// TIA Portal project "SimpleProject" (V17)

(* hardware
DEVICE "PLC_1"  S7-1200 Station
   slot 0: "Rack_0"  S7-1200 Rack  Rack  V1.0
   slot 1: "PLC_1"  CPU 1214C AC/DC/Rly  6ES7 214-1BG40-0XB0  V4.5
*)

// ===== PLC "PLC_1"  CPU 1214C AC/DC/Rly =====

VAR_GLOBAL   // PLC tag table "MotorControl"
   "Start" AT %I0.0 : Bool;
   "Stop" AT %I0.1 : Bool;
   "Motor" AT %Q0.0 : Bool;
END_VAR

FUNCTION "MotorControl" : Void   // FC1, LAD
{ S7_Optimized_Access := 'TRUE' }
VERSION : 0.1
BEGIN

REGION Network 1
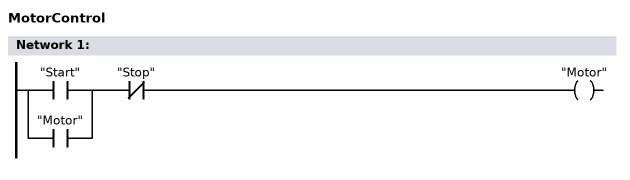
   RUNG wire#powerrail
      Contact( "Start" )
      wire#w1
      I_Contact( "Stop" )
      Coil( "Motor" )
   END_RUNG
   RUNG wire#powerrail
      Contact( "Motor" )
   END_RUNG wire#w1
   // the same network as SCL:
   "Motor" := ("Start" OR "Motor") AND NOT "Stop";
END_REGION
END_FUNCTION

ORGANIZATION_BLOCK "Main"   // OB1, LAD, ProgramCycle
TITLE = "Main Program Sweep (Cycle)"
{ S7_Optimized_Access := 'TRUE' }
VERSION : 0.1
   VAR_INPUT
      Initial_Call : Bool;   // Initial call of this OB
      Remanence : Bool;   // =True, if remanent data are available
   END_VAR
BEGIN
END_ORGANIZATION_BLOCK